(* Logix 5000 project; controller ECE119L_Elevator 5069-L306ERM rev 32.11; software revision 32.01 *)

TASK MainTask (continuous, watchdog 500 ms) : MainProgram

MODULES
   Local : 5069-L306ERM (5069 0, rev 32.11)
      VFD : PowerFlex 525-EENET (Ethernet 192.168.1.15, rev 5.1, Output RPI 20 ms)
      SERVO : vendor 1 type 37 code 46 (Ethernet 192.168.1.1, rev 7.1, MotionDiagnostics RPI 1 ms, MotionSync RPI 1 ms)
      Digital_In : vendor 1 type 7 code 391 (5069 1, rev 2.1, StandardDataDriven RPI 5 ms)
      Digital_Out : 5069-OB16 (5069 2, rev 2.1, StandardDataDriven RPI 5 ms)
      Analog_In1 : vendor 1 type 115 code 314 (5069 3, rev 2.1, StandardDataDriven RPI 100 ms)
      Analog_In2 : vendor 1 type 115 code 314 (5069 4, rev 2.1, StandardDataDriven RPI 100 ms)
      Analog_Out : vendor 1 type 115 code 320 (5069 5, rev 2.1, StandardDataDriven RPI 80 ms)
END_MODULES

VAR_GLOBAL   (* controller tags *)
   Axis_1 : AXIS_CIP_DRIVE;
   Blue_Butt : ALIAS FOR Local:1:I.Pt10.Data;
   Blue_LED : ALIAS FOR Local:2:O.Pt10.Data;
   Blue_SW : ALIAS FOR Local:1:I.Pt14.Data;
   FLOOR_1 : ALIAS FOR Local:1:I.Pt00.Data;
   FLOOR_1_LED : ALIAS FOR Local:2:O.Pt00.Data;
   FLOOR_2 : ALIAS FOR Local:1:I.Pt01.Data;
   FLOOR_2_LED : ALIAS FOR Local:2:O.Pt01.Data;
   FLOOR_3 : ALIAS FOR Local:1:I.Pt02.Data;
   FLOOR_3_LED : ALIAS FOR Local:2:O.Pt02.Data;
   FLOOR_4 : ALIAS FOR Local:1:I.Pt03.Data;
   FLOOR_4_LED : ALIAS FOR Local:2:O.Pt03.Data;
   Green_Butt : ALIAS FOR Local:1:I.Pt08.Data;
   Green_LED : ALIAS FOR Local:2:O.Pt08.Data;
   Green_SW : ALIAS FOR Local:1:I.Pt12.Data;
   Knob : ALIAS FOR Local:4:I.Ch00.Data;
   LCD : ALIAS FOR Local:5:O.Ch00.Data;
   M_Group : MOTION_GROUP;
   OUT_5V : ALIAS FOR Local:2:O.Pt07.Data;
   Red_Butt : ALIAS FOR Local:1:I.Pt11.Data;
   Red_LED : ALIAS FOR Local:2:O.Pt11.Data;
   Red_SW : ALIAS FOR Local:1:I.Pt15.Data;
   Round_Knob : INT;
   Yellow_Butt : ALIAS FOR Local:1:I.Pt09.Data;
   Yellow_LED : ALIAS FOR Local:2:O.Pt09.Data;
   Yellow_SW : ALIAS FOR Local:1:I.Pt13.Data;
END_VAR

PROGRAM MainProgram   (* main routine MainRoutine *)

ROUTINE MainRoutine   (* ladder *)
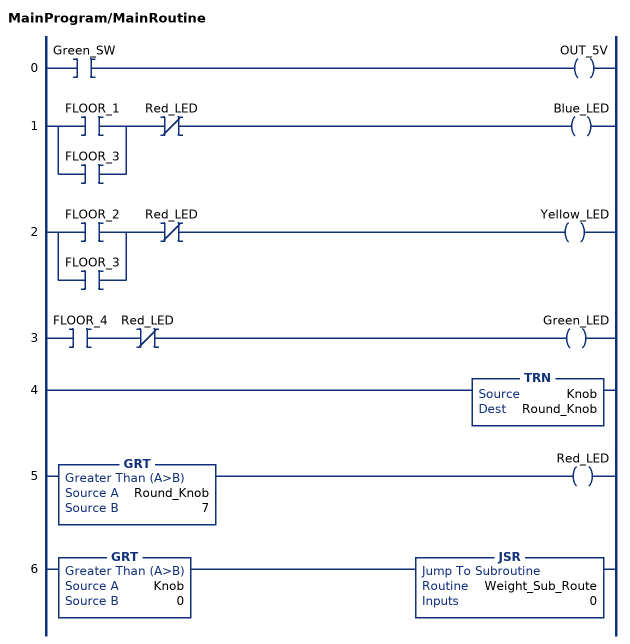
   0: XIC(Green_SW)OTE(OUT_5V);
   1: [XIC(FLOOR_1) ,XIC(FLOOR_3) ]XIO(Red_LED)OTE(Blue_LED);
   2: [XIC(FLOOR_2) ,XIC(FLOOR_3) ]XIO(Red_LED)OTE(Yellow_LED);
   3: XIC(FLOOR_4)XIO(Red_LED)OTE(Green_LED);
   4: TRN(Knob,Round_Knob);
   5: GRT(Round_Knob,7)OTE(Red_LED);
   6: GRT(Knob,0)JSR(Weight_Sub_Route,0);
END_ROUTINE

ROUTINE Weight_Sub_Route   (* structured text *)
   case Round_Knob of
   	0: LCD:=0.000000;
   	1: LCD:=1.002000;
   	2: LCD:=2.002000;
   	3: LCD:=3.002000;
   	4: LCD:=4.003000;
   	5: LCD:=5.003000;
   	6: LCD:=6.003000;
   	7: LCD:=7.003500;
   	8: LCD:=8.004000;
   	9: LCD:=9.004000;
   	10: LCD:=10.004000;
   	ELSE
   		LCD:=Round_Knob;
   end_case;
END_ROUTINE
END_PROGRAM
